TYPE STR :
STRUCT
		MesIdc			: REAL;   						(* (A) DC current *)
		MesUdc			: REAL;							(* (V) DC voltage *)
END_STRUCT
END_TYPE

(* stored: Version 1.1.0.1, ProductVersion 3.1.4024.9
   DUT STR: Id {3b877ebf-7a65-4916-96e9-6019742f5ba8} *)
